(* CODESYS project Networkvariables.sender.20190701.project
   Description: This example demonstrates how to share a variable within a network. One application is sending the variable and the other one receives it.
   Version: 1.0.0.0
   Title: Network Variables
   Company: 3S - Smart Software Solutions GmbH

Project tree, tasks and I/O mapping:
  Sender : Changsha-Cyber-MI-linux, Changsha Cyber-MI Co., Ltd., version 3.5.10.40
    application App_Send
      libraries: Standard, * (System)
      task Task (cyclic, interval t#20ms, priority 1) calls Main_Send
      global variables NVL_sender
      program Main_Send [ST]
    SoftMotion General Axis Pool
*)

// Sender/App_Send/NVL_sender
{attribute 'qualified_only'}
VAR_GLOBAL
	iglobvar:INT; 
	bGlobVar01:BOOL;
	uGlobVar03:UINT;
	uGlobVar04:UINT;
	uGlobVar05:UINT;
	uiVar07:UINT;
END_VAR

// Sender/App_Send/Main_Send
PROGRAM Main_Send
VAR
	TxDiag : NetVarUdp.NetVarUDPDiagStruct;
END_VAR

nvl_sender.iglobvar := nvl_sender.iglobvar + 1;

(* Diagnostic *)
TxDiag := NetVar_App_Send_GVL.NetVarTxDiag_UDP[0];

END_PROGRAM
